// TIA Portal V19 export
FUNCTION_BLOCK "RMP_FRQ_SPD"   // FB11, LAD
TITLE = RMP Sinamics speed & torque control
{ S7_Optimized_Access := 'TRUE' }
AUTHOR : Joni_Lahtonen
FAMILY : Raumaster_Paper
VERSION : 1.0
// This block uses profidrive profile to control siemens frequency converters.
// Use communication profile 352 (6/6) in HW configuration.
// stored: MemoryReserve 100, SetENOAutomatically false
   VAR_INPUT
      Fwd { ExternalAccessible := 'False'; ExternalVisible := 'False'; ExternalWritable := 'False'} : Bool;   // Drive forward request / Eteen käsky
      Rev { ExternalAccessible := 'False'; ExternalVisible := 'False'; ExternalWritable := 'False'} : Bool;   // Drive reverse request / Taakse käsky
      Invert : Bool;   // Invert drive rotation direction / Ajosuunnan muutos
      Ack { ExternalAccessible := 'False'; ExternalVisible := 'False'; ExternalWritable := 'False'} : Bool;   // Drive alarm acknowledge / Häiriönkuittaus
      Speed_req { ExternalAccessible := 'False'; ExternalVisible := 'False'; ExternalWritable := 'False'} : Real;   // Drive speed request 100.0 = 3000rpm / Nopeusohje
      Torque_req { ExternalAccessible := 'False'; ExternalVisible := 'False'; ExternalWritable := 'False'} : Real;   // Drive torque request 100.0 = 100% / Momenttiohje
      Address { ExternalAccessible := 'False'; ExternalVisible := 'False'; ExternalWritable := 'False'} : HW_IO;   // Drive telegram HW address / HW-osoite
      "Type" { ExternalAccessible := 'False'; ExternalVisible := 'False'; ExternalWritable := 'False'} : Bool;   // Drive type 0 = Siemens / 1 = ABB / 0 = Siemens / 1 = ABB
   END_VAR
   VAR_OUTPUT
      Status { ExternalAccessible := 'False'; ExternalVisible := 'False'; ExternalWritable := 'False'} : Word;   // Drive status / Taajuusmuuttajan tilasana
      Speed_CV { ExternalAccessible := 'False'; ExternalVisible := 'False'; ExternalWritable := 'False'} : Real;   // Drive actual speed 100.0 = 3000rpm / Nopeuden oloarvo
      Torque_CV { ExternalAccessible := 'False'; ExternalVisible := 'False'; ExternalWritable := 'False'} : Real;   // Drive actual torgue 100.0 = 100% / Momentin oloarvo
      Run_fwd { ExternalAccessible := 'False'; ExternalVisible := 'False'; ExternalWritable := 'False'} : Bool;   // Drive is running forward / Käy eteen
      Run_rev { ExternalAccessible := 'False'; ExternalVisible := 'False'; ExternalWritable := 'False'} : Bool;   // Drive is running reverse / Käy taakse
      Alarm { ExternalAccessible := 'False'; ExternalVisible := 'False'; ExternalWritable := 'False'} : Bool;   // Drive alarm on / Häiriö päällä
      Alarm_number { ExternalAccessible := 'False'; ExternalVisible := 'False'; ExternalWritable := 'False'} : Int;   // Drive alarm number / Häiriönumero
   END_VAR
   VAR
      Alarm_delay { S7_SetPoint := 'True'} : TON_TIME;
   END_VAR
   VAR_TEMP
      Return_value : Int;
      Siemens : Struct
         In : Struct
            SW : Struct
               Set_point : Bool;   // Setpoint / actual value deviation within the tolerancerange.
               Mst_control_req : Bool;   // The automation system is requested to accept the invertercontrol.
               F_reached : Bool;   // Speed is greater than or equal to the corresponding
               Motor_current_limit : Bool;
               Brake : Bool;
               Motor_overload : Bool;
               CW_CCW_rotation : Bool;
               Converter_overload : Bool;
               Ready_for_on : Bool;   // Power supply switched on; electronics initialized; pulses
               Ready_to_run : Bool;
               Oper_enabled : Bool;   // Motor follows setpoint. See control word 1, bit 3.
               Fault_active : Bool;   // The inverter has a fault. Acknowledge fault using STW1.7.
               OFF2_status : Bool;   // Coast down to standstill is not active.
               OFF3_status : Bool;   // Quick stop is not active.
               Start_lockout : Bool;   // It is only possible to switch on the motor after an OFF1followed by ON.
               Alarm_active : Bool;   // Motor remains switched on; no acknowledgement isnecessary.
            END_STRUCT;
            Speed_CV : Int;
            Data_2 : Int;
            Torque_CV : Int;
            Alarm_nbr : Int;
            Data5 : Int;
         END_STRUCT;
         Out : Struct
            CW : Struct
               Jog_left : Bool;
               Jog_right : Bool;
               Setp_valid : Bool;
               Setp_invert : Bool;
               NC1 : Bool;
               Mop_up : Bool;
               Mop_dn : Bool;
               NC2 : Bool;
               On_Off1 : Bool;   // The motor brakes with the ramp-down time p1121 of theramp-function generator. The inverter switches off the motorat standstill.
               OFF2 : Bool;   // Switch off the motor immediately, the motor then coasts
               OFF3 : Bool;   // Quick stop: The motor brakes with the OFF3 ramp-down
               Oper : Bool;   // Immediately switch-off motor (cancel pulses).
               Cond : Bool;   // The inverter immediately sets its ramp-function generatoroutput to 0.
               Enable_RFG : Bool;   // The output of the ramp-function generator stops at the actualvalue.
               Enable_setpoint : Bool;   // Motor accelerates with the ramp-up time p1120 to thesetpoint
               Ack_fault : Bool;   // Acknowledge fault. If the ON command is still active, theinverter switches to"closing lockout" state.
            END_STRUCT;
            Speed_req : Int;
            Torque_req_p : Int;
            Torque_req_m : Int;
            Data5 : Int;
            Data6 : Int;
         END_STRUCT;
      END_STRUCT;
      ABB : Struct
         In : Struct
            SW : Struct
               At_setpoint : Bool;   // Setpoint / actual value deviation within the tolerancerange. / Actual value equals reference
               Remote : Bool;   // The automation system is requested to accept the invertercontrol. / Drive control location: REMOTE (EXT1 or EXT2)
               Above_limit : Bool;   // Speed is greater than or equal to the corresponding / Actual frequency or speed equals or exceeds supervision limit
               Res_1 : Bool;
               Brake : Bool;   // Brake if parametrized
               Res_3 : Bool;
               Res_4 : Bool;
               FBA_Error : Bool;
               Ready_on : Bool;   // Power supply switched on; electronics initialized; pulses / Ready to switch on
               Ready_run : Bool;   // Ready to operate
               Ready_ref : Bool;   // Motor follows setpoint. See control word 1, bit 3. / Operation enabled
               Tripped : Bool;   // The inverter has a fault. Acknowledge fault using STW1.7. / Fault
               OFF2_status : Bool;   // Coast down to standstill is not active. / OFF 2 inactive
               OFF3_status : Bool;   // Quick stop is not active. / OFF 3 inactive
               Switch_on_inhib : Bool;   // It is only possible to switch on the motor after an OFF1followed by ON. / Switch on inhibited
               Warning : Bool;   // Motor remains switched on; no acknowledgement isnecessary. / Alarm / warning active
            END_STRUCT;
            Speed_CV : Int;
            Data_2 : Int;
            Torque_CV : Int;
            Alarm_nbr : Int;
            Data5 : Int;
         END_STRUCT;
         Out : Struct
            CW : Struct
               Res_1 : Bool;
               Res_2 : Bool;
               Remote_cmd : Bool;
               Ext_ctrl_loc : Bool;
               Res_4 : Bool;
               Res_5 : Bool;
               Res_6 : Bool;
               Res_7 : Bool;
               OFF1_Control : Bool;   // The motor brakes with the ramp-down time p1121 of theramp-function generator. The inverter switches off the motorat standstill.
               OFF2_Control : Bool;   // Switch off the motor immediately, the motor then coasts
               OFF3_Control : Bool;   // Quick stop: The motor brakes with the OFF3 ramp-down
               Inhibit_oper : Bool;   // Immediately switch-off motor (cancel pulses).
               Ramp_out_zero : Bool;   // The inverter immediately sets its ramp-function generatoroutput to 0.
               Ramp_hold : Bool;   // The output of the ramp-function generator stops at the actualvalue.
               Ramp_in_zero : Bool;   // Motor accelerates with the ramp-up time p1120 to thesetpoint
               Reset : Bool;   // Acknowledge fault. If the ON command is still active, theinverter switches to"closing lockout" state.
            END_STRUCT;
            Speed_req : Int;
            Torque_req_p : Int;
            Torque_req_m : Int;
            Data5 : Int;
            Data6 : Int;
         END_STRUCT;
      END_STRUCT;
      Speed_R : Real;
      Torque_R : Real;
      Current_R : Real;
      Speed_req_R : Real;
      Torque_req_R : Real;
      Temp_int : Int;
      Temp_word : Word;
      Error_b : Bool;
      Fwd_req : Bool;
      Setp_invert : Bool;
   END_VAR
BEGIN

REGION Network 1 (SCL): Nopeusohje
   //=========================================================================
   // Raumaster Paper Oy
   // (c)Copyright 2018 All Rights Reserved
   //-----------------------------------------------------------------------------
   // Library: RmpLib
   // Tested with: S7-1516F-3PN/DP V2.1
   //              G120 
   // Engineering: TIA Portal V15
   // Restrictions: 
   // Requirements: S7-1200 / S7-1500
   // Functionality:   This block is made for controlling Siemens drives
   //                  trough Profidrive profile.
   //                  Block uses Siemens telegram 352 6 word in / 6 words out
   //=========================================================================



   IF NOT #Type THEN

       REGION Siemens drive

           //Initialize local variables
           #Siemens.Out.Speed_req := 0;
           #Siemens.Out.Torque_req_p := 0;
           #Temp_word := 0;
           SCATTER(IN := #Temp_word,
                   OUT => #Siemens.Out.CW);

           //Read drive data
           #Return_value := DPRD_DAT(LADDR := #Address, RECORD => #Siemens);

           //Drive status word
           GATHER(IN := #Siemens.In.SW, OUT => #Status);

           #Speed_CV := ABS(INT_TO_REAL(#Siemens.In.Speed_CV) / 16.384);
           #Torque_CV := ABS(INT_TO_REAL(#Siemens.In.Torque_CV) / 16.384);


           //Drive alarm active
           #Alarm_number := #Siemens.In.Alarm_nbr;
           #Alarm_delay(IN := #Siemens.In.SW.Fault_active,
           PT := T#100ms,
           Q => #Alarm);

           //Drive running forward
           #Run_fwd := #Siemens.In.SW.Oper_enabled AND ((NOT #Siemens.In.SW.CW_CCW_rotation AND NOT #Invert) OR (#Siemens.In.SW.CW_CCW_rotation AND #Invert));

           //Drive running reverse
           #Run_rev := #Siemens.In.SW.Oper_enabled AND ((#Siemens.In.SW.CW_CCW_rotation AND NOT #Invert) OR (NOT #Siemens.In.SW.CW_CCW_rotation AND #Invert));

           //Set control bits
           #Siemens.Out.CW.OFF2 := true;
           #Siemens.Out.CW.Oper := true;
           #Siemens.Out.CW.Cond := true;
           #Siemens.Out.CW.Enable_RFG := true;
           #Siemens.Out.CW.Enable_setpoint := true;
           #Siemens.Out.CW.Setp_valid := true;
           #Siemens.Out.CW.OFF3 := true;

           //Drive forward request
           #Fwd_req := (#Fwd OR #Rev) AND #Siemens.In.SW.Ready_for_on AND #Siemens.In.SW.OFF3_status AND NOT #Siemens.In.SW.Fault_active AND NOT #Error_b;

           //Drive forward command
           #Siemens.Out.CW.On_Off1 := #Fwd_req;

           //Drive reverse command
           #Setp_invert := ((#Invert AND NOT #Rev) OR (NOT #Invert AND #Rev)) AND #Fwd_req;

           //Fault ack from drive
           #Siemens.Out.CW.Ack_fault := #Ack;

           //Speed request for drive
           IF #Fwd_req AND NOT #Setp_invert THEN
               #Siemens.Out.Speed_req := REAL_TO_INT(ABS(#Speed_req * 16.384));
           ELSIF #Fwd_req AND #Setp_invert THEN
               #Siemens.Out.Speed_req := - REAL_TO_INT(ABS(#Speed_req * 16.384));
           ELSE
               #Siemens.Out.Speed_req := 0;
           END_IF;


           //Torque request for drive, max positive torque
           #Siemens.Out.Torque_req_p := REAL_TO_INT(#Torque_req * 16.384);
           #Siemens.Out.Torque_req_m := - #Siemens.Out.Torque_req_p;


           //Write drive data
           #Return_value := DPWR_DAT(LADDR := #Address, RECORD := #Siemens.Out);

       END_REGION

   ELSE

       REGION ABB Drive

           //Initialize local variables
           #ABB.Out.Speed_req := 0;
           #ABB.Out.Torque_req_p := 0;
           #Temp_word := 0;
           SCATTER(IN := #Temp_word, OUT => #ABB.Out.CW);

           //Read drive data
           #Return_value := DPRD_DAT(LADDR := #Address, RECORD => #ABB.In);

           //Drive status word
           GATHER(IN := #ABB.In.SW,OUT => #Status);

           #Speed_CV := ABS(INT_TO_REAL(#ABB.In.Speed_CV) / 20.0);
           #Torque_CV := ABS(INT_TO_REAL(#ABB.In.Torque_CV) / 20.0);


           //Drive alarm active
           #Alarm_number := #ABB.In.Alarm_nbr;
           #Alarm_delay(IN := #ABB.In.SW.Tripped, PT := T#200ms, Q => #Alarm);

           //Drive running forward
           #Run_fwd := #ABB.In.SW.Ready_ref AND ((#ABB.In.Speed_CV > 0 AND NOT #Invert) OR (#ABB.In.Speed_CV < 0 AND #Invert));

           //Drive running reverse
           #Run_rev := #ABB.In.SW.Ready_ref AND ((#ABB.In.Speed_CV < 0 AND NOT #Invert) OR (#ABB.In.Speed_CV > 0 AND #Invert));

           //Set control bits
           #ABB.Out.CW.OFF1_Control := #ABB.In.SW.Ready_on;
           #ABB.Out.CW.OFF2_Control := true;
           #ABB.Out.CW.OFF3_Control := true;
           #ABB.Out.CW.Ramp_out_zero := true;
           #ABB.Out.CW.Ramp_hold := true;
           #ABB.Out.CW.Ramp_in_zero := true;
           #ABB.Out.CW.Remote_cmd := true;


           //Drive forward request
           #Fwd_req := (#Fwd OR #Rev) AND NOT #ABB.In.SW.Tripped;// AND #ABB.In.SW.Ready_on AND #ABB.In.SW.OFF3_status

           //Drive forward command
           #ABB.Out.CW.Inhibit_oper := #Fwd_req;

           //Drive reverse command
           #Setp_invert := ((#Invert AND NOT #Rev) OR (NOT #Invert AND #Rev)) AND #Fwd_req;

           //Fault ack from drive
           #ABB.Out.CW.Reset := #Ack;

           //Speed request for drive
           IF #Fwd_req AND NOT #Setp_invert THEN
               #ABB.Out.Speed_req := REAL_TO_INT(ABS(#Speed_req * 20.0));
           ELSIF #Fwd_req AND #Setp_invert THEN
               #ABB.Out.Speed_req := - REAL_TO_INT(ABS(#Speed_req * 20.0));
           ELSE
               #ABB.Out.Speed_req := 0;
           END_IF;

           #ABB.Out.Torque_req_p := REAL_TO_INT(#Torque_req * 20.0);
           #ABB.Out.Torque_req_m := - #ABB.Out.Torque_req_p;

           //Write drive data
           #Return_value := DPWR_DAT(LADDR := #Address, RECORD := #ABB.Out);

       END_REGION
   END_IF;
END_REGION
END_FUNCTION_BLOCK
